// TIA Portal V17 export
// export: Created 2022-04-06T07:28:39.4284423Z, ExportSetting WithDefaults, DisplayName Totally Integrated Automation Portal, DisplayVersion V17, DisplayName TIA Portal Openness, DisplayVersion V17, DisplayName TIA Portal Version Control Interface, DisplayVersion V17, DisplayName TIA Portal Test Suite Advanced, DisplayVersion V17, DisplayName SINAMICS Startdrive Advanced, DisplayVersion V17, DisplayName SINAMICS Startdrive G130, G150, S120, S150, SINAMICS MV, S210, DisplayVersion V17, DisplayName SINAMICS Startdrive G110M, G120, G120C, G120D, G120P, G115D, DisplayVersion V17, DisplayName STEP 7 Professional, DisplayVersion V17, DisplayName STEP 7 Safety, DisplayVersion V17, DisplayName WinCC Advanced / Unified PC, DisplayVersion V17
FUNCTION_BLOCK "FileHandling"   // FB4, LAD
{ S7_Optimized_Access := 'TRUE' }
VERSION : 0.1
// stored: AutoNumber true, IsIECCheckEnabled true, IsRetainMemResEnabled false, MemoryReserve 100, SetENOAutomatically false, UDAEnableTagReadback false
   VAR
      instFileWriteC_SFB { S7_SetPoint := 'True'} : FileWriteC;
      instFileReadC_SFB { S7_SetPoint := 'True'} : FileReadC;
      instFileDelete { S7_SetPoint := 'True'} : FileDelete;
      statData { S7_SetPoint := 'True'} : Array[0..3] of Byte;
   END_VAR
BEGIN

REGION Network 1
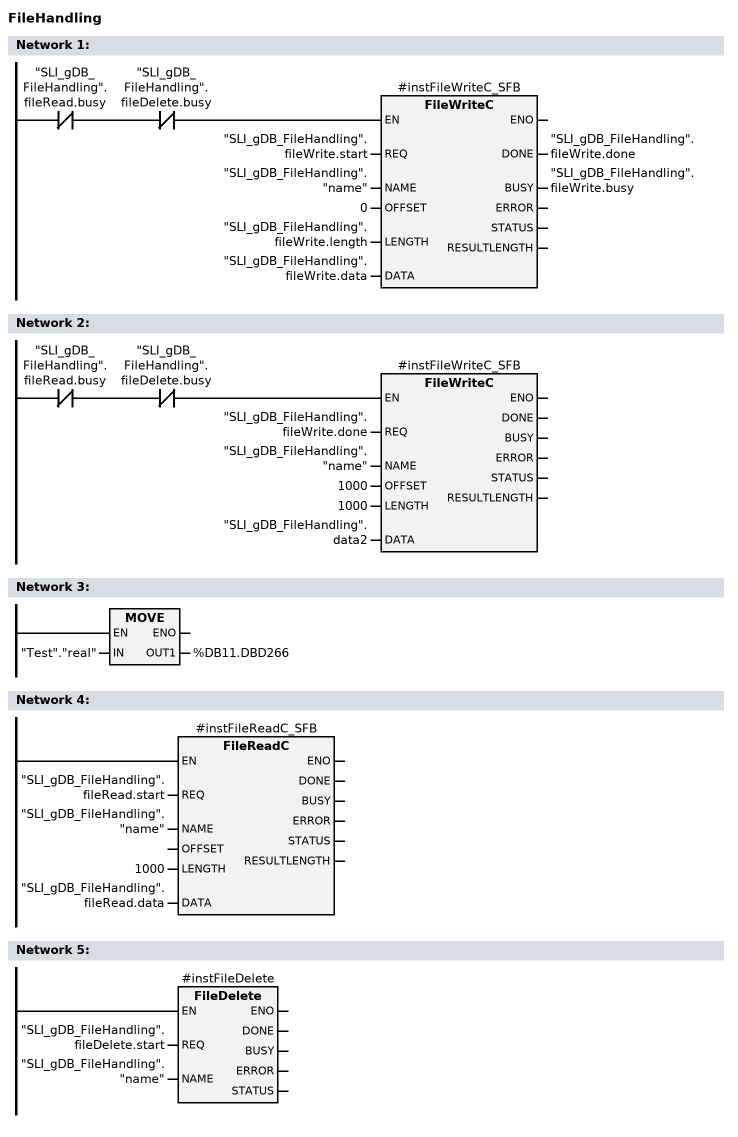
   RUNG wire#powerrail
      I_Contact( "SLI_gDB_FileHandling".fileRead.busy )
      I_Contact( "SLI_gDB_FileHandling".fileDelete.busy )
      #instFileWriteC_SFB.FileWriteC(REQ := "SLI_gDB_FileHandling".fileWrite.start, "Name" := "SLI_gDB_FileHandling"."name", Offset := 0, Length := "SLI_gDB_FileHandling".fileWrite.length, Data := "SLI_gDB_FileHandling".fileWrite.data, Done => "SLI_gDB_FileHandling".fileWrite.done, Busy => "SLI_gDB_FileHandling".fileWrite.busy, Error =>, Status =>, ResultLength =>)
   END_RUNG
   // the same network as SCL:
   IF NOT "SLI_gDB_FileHandling".fileRead.busy AND NOT "SLI_gDB_FileHandling".fileDelete.busy THEN
       #instFileWriteC_SFB(REQ := "SLI_gDB_FileHandling".fileWrite.start,   // FileWriteC
                           "Name" := "SLI_gDB_FileHandling"."name",
                           Offset := 0,
                           Length := "SLI_gDB_FileHandling".fileWrite.length,
                           Data := "SLI_gDB_FileHandling".fileWrite.data,
                           Done => "SLI_gDB_FileHandling".fileWrite.done,
                           Busy => "SLI_gDB_FileHandling".fileWrite.busy);
   END_IF;
END_REGION

REGION Network 2
   RUNG wire#powerrail
      I_Contact( "SLI_gDB_FileHandling".fileRead.busy )
      I_Contact( "SLI_gDB_FileHandling".fileDelete.busy )
      #instFileWriteC_SFB.FileWriteC(REQ := "SLI_gDB_FileHandling".fileWrite.done, "Name" := "SLI_gDB_FileHandling"."name", Offset := 1000, Length := 1000, Data := "SLI_gDB_FileHandling".data2, Done =>, Busy =>, Error =>, Status =>, ResultLength =>)
   END_RUNG
   // the same network as SCL:
   IF NOT "SLI_gDB_FileHandling".fileRead.busy AND NOT "SLI_gDB_FileHandling".fileDelete.busy THEN
       #instFileWriteC_SFB(REQ := "SLI_gDB_FileHandling".fileWrite.done,   // FileWriteC
                           "Name" := "SLI_gDB_FileHandling"."name",
                           Offset := 1000,
                           Length := 1000,
                           Data := "SLI_gDB_FileHandling".data2);
   END_IF;
END_REGION

REGION Network 3
   RUNG wire#powerrail
      Move(in := "Test"."real", out1 => %DB11.DBD266)
   END_RUNG
   // the same network as SCL:
   %DB11.DBD266 := "Test"."real";
END_REGION

REGION Network 4
   RUNG wire#powerrail
      #instFileReadC_SFB.FileReadC(REQ := "SLI_gDB_FileHandling".fileRead.start, "Name" := "SLI_gDB_FileHandling"."name", Offset :=, Length := 1000, Data := "SLI_gDB_FileHandling".fileRead.data, Done =>, Busy =>, Error =>, Status =>, ResultLength =>)
   END_RUNG
   // the same network as SCL:
   #instFileReadC_SFB(REQ := "SLI_gDB_FileHandling".fileRead.start,   // FileReadC
                      "Name" := "SLI_gDB_FileHandling"."name",
                      Length := 1000,
                      Data := "SLI_gDB_FileHandling".fileRead.data);
END_REGION

REGION Network 5
   RUNG wire#powerrail
      #instFileDelete.FileDelete(REQ := "SLI_gDB_FileHandling".fileDelete.start, "Name" := "SLI_gDB_FileHandling"."name", Done =>, Busy =>, Error =>, Status =>)
   END_RUNG
   // the same network as SCL:
   #instFileDelete(REQ := "SLI_gDB_FileHandling".fileDelete.start, "Name" := "SLI_gDB_FileHandling"."name");   // FileDelete
END_REGION
END_FUNCTION_BLOCK
